{attribute 'qualified_only'}
{attribute 'strict'}
TYPE STATES :
(
	enum_member := 0
);
END_TYPE

(* stored: Version 1.1.0.1, ProductVersion 3.1.4020.3
   DUT STATES: Id {63992934-0974-4bf2-a86c-1001741663c9} *)
